FUNCTION_BLOCK FB_EnclosureConditioningSFC
VAR_IN_OUT
	//IPSState					:	ST_InternalPowerStatus;
	IPSDemand					:	ST_PowerDemand;
	ConditioningRequirements	: 	ST_ConditioningRequirements;
	Control							:	ST_CoolingSystem_Control;
	Get							:	ST_CoolingSystemGet;	
END_VAR

VAR_OUTPUT
	SFCCurrentStep	:	STRING;
END_VAR
VAR_OUTPUT
	SFCActive	:	BOOL;
END_VAR

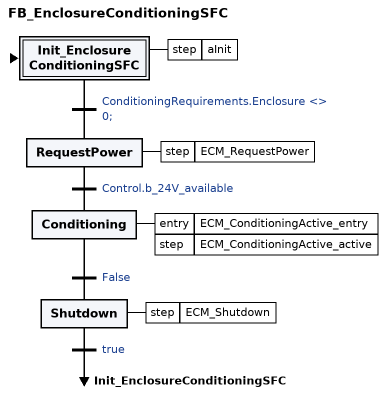
INITIAL_STEP Init_EnclosureConditioningSFC:
    aInit(N);  // step action
END_STEP
TRANSITION FROM Init_EnclosureConditioningSFC TO RequestPower
    := ConditioningRequirements.Enclosure <> 0;
END_TRANSITION
STEP RequestPower:
    ECM_RequestPower(N);  // step action
END_STEP
TRANSITION FROM RequestPower TO Conditioning
    := Control.b_24V_available;
END_TRANSITION
STEP Conditioning:
    ECM_ConditioningActive_entry(P1);  // entry action
    ECM_ConditioningActive_active(N);  // step action
END_STEP
TRANSITION FROM Conditioning TO Shutdown
    := False;
END_TRANSITION
STEP Shutdown:
    ECM_Shutdown(N);  // step action
END_STEP
TRANSITION FROM Shutdown TO Init_EnclosureConditioningSFC
    := true;
END_TRANSITION

ACTION aInit:
SFCActive := False;
END_ACTION

ACTION ECM_ConditioningActive_active:
IF ConditioningRequirements.Enclosure = 0 THEN
	SFCTip := TRUE;
END_IF
END_ACTION

ACTION ECM_ConditioningActive_entry:
Control.b_CloseBatteryLoopValve 	:= 	FALSE;
Control.b_CloseFancoilLoopValve 	:= 	FALSE;
Control.b_CloseInverterLoopValve := 	TRUE;

Control.b_DCFancoilEnable 		:= TRUE;
Control.b_DCPumpEnable 			:= TRUE;
END_ACTION

ACTION ECM_RequestPower:
SFCActive:= True;
IPSDemand.b_Demand_24V := TRUE;
END_ACTION

ACTION ECM_Shutdown:
Control.b_CloseBatteryLoopValve 	:= 	FALSE;
Control.b_CloseFancoilLoopValve 	:= 	FALSE;
Control.b_CloseInverterLoopValve := 	FALSE;

Control.b_DCFancoilEnable 		:= 	FALSE;
Control.b_DCPumpEnable 			:= 	FALSE;

IPSDemand.b_Demand_24V 		:= 	FALSE;
SFCActive:= False;
END_ACTION

METHOD SFCEnable : BOOL
VAR_INPUT
	Enable	:	Bool;
END_VAR
IF Enable THEN
	SFCInit := FALSE;
ELSE
	SFCActive:= FALSE;
	SFCInit := TRUE;
END_IF
END_METHOD

END_FUNCTION_BLOCK

(* stored: Version 1.1.0.1, ProductVersion 3.1.4024.12
   POU FB_EnclosureConditioningSFC: Id {30c2efd6-cdbc-4ba3-b10c-9309fd99d802}, SpecialFunc None
   Action aInit: Id {c9524e06-9238-41fd-b4ce-9e7b84cbc60e}
   Action ECM_ConditioningActive_active: Id {4d868abc-3432-4aeb-9e14-70a8c25dec67}
   Action ECM_ConditioningActive_entry: Id {f03e303d-dc01-4aff-97ca-384044b59d18}
   Action ECM_RequestPower: Id {1429f80a-c7be-4fcd-b944-cbef3f8ccac8}
   Action ECM_Shutdown: Id {cccade72-8dd1-442a-8d85-50be43acb559}
   Method SFCEnable: Id {250c9ecf-0fff-4489-94fb-141288788bcf} *)
